// Stepwise homing process
CASE nTestStep OF
    0: // Await full power-up, start first stage home
        IF fbPower[4].PowerIsEnabled THEN
			 fbHome.Home(
					Position := fExpectedPosition,
					BufferMode := MC_BufferMode.MC_Aborting,
					HomeMode:=E_EpicsHomeCmd.HOME_VIA_HIGH
			);
            nTestStep := 1;
        END_IF
    1: // Simulate Forward Limit pulse (stage 1 complete)
        IF fbCamSwitchPulserSearch.Q THEN
            fbLimSwStatus[4].LimitForwardEnable := FALSE;
            fbCamSwitchPulserSearch.IN := FALSE;
            fbCamSwitchPulserSync.IN := TRUE;
            nTestStep := 2;
        END_IF
    2: // Release Forward Limit (simulate rising edge)
        IF fbCamSwitchPulserSync.Q THEN
            fbLimSwStatus[4].LimitForwardEnable := TRUE;
            nTestStep := 3;
        END_IF
    3: // When forward limit home is done, prepare for the home switch
        IF fbHome.LimHomeDone THEN
            fbCamSwitchPulserSearch.IN := TRUE;
            fbCamSwitchPulserSync.IN := FALSE;
            nTestStep := 4;
        END_IF
    4: // Simulate Home switch pulse
        IF fbCamSwitchPulserSearch.Q THEN
            fbLimSwStatus[4].LimitHome := TRUE;
            fbCamSwitchPulserSearch.IN := FALSE;
            fbCamSwitchPulserSync.IN := TRUE;
            nTestStep := 5;
        END_IF
    5: // Release Home switch
        IF fbCamSwitchPulserSync.Q THEN
            fbLimSwStatus[4].LimitHome := FALSE;
            nTestStep := 6;
        END_IF
    6: // Wait for homing full completion
        IF fbHome.Done THEN
            nTestStep := 7;
        END_IF
END_CASE

// Cyclic calls required for simulation and status updates
fbPower[4]();
fbHome();
fbCamSwitchPulserSearch();
fbCamSwitchPulserSync();
fbTestTimer();

// Finish test if homing is complete (step 7), or timeout
IF nTestStep = 7 THEN
    bCalibrated := fbHome.Done;
    AssertEquals_BOOL(
        Expected := TRUE,
        Actual := fbAxisRef[4].Status.Homed,
        Message := 'Axis not calibrated #1'
    );
    AssertEquals_LREAL(
        Delta := 0.001,
        Expected := fExpectedPosition,
        Actual := fbAxisRef[4].NcToPlc.ActPos,
        Message := 'Position is not the expected #2'
    );
    TEST_FINISHED();

ELSIF fbTestTimer.Q THEN
    AssertTrue(
        Condition := FALSE,
        Message := CONCAT('Timed out at step: ', TO_STRING(nTestStep))
    );
    TEST_FINISHED();
END_IF
END_METHOD

METHOD PRIVATE GivenHomeCmdHomeViaLowModeAndHomeSwPulseThenMoveToUserDefineOffset_Test5
VAR_INST
    fbHome : FB_HomeNC(
		AxisRef:=fbAxisRef[5],
		iLimSwStatus:=fbLimSwStatus[5],
		iMotionLogger:=fbMotionLogger[5]
	) := ( Mode := E_EpicsHomeCmd.HOME_VIA_LOW );
	
    fbTestTimer: TON := (IN:=TRUE, PT:=T#5S);
    fbCamSwitchPulserSearch: TON := (IN:=TRUE, PT:=T#500MS);
    fbCamSwitchPulserSync: TON := (PT:=T#1000MS);
    nTestStep : INT;
    fExpectedPosition : LREAL := 20.0;
    fActPosition : LREAL;
	bCalibrated: BOOL;
    // reset this when error or homeDone
    bHomingOverride : BOOL := TRUE;

END_VAR
TEST(__POUNAME());

// Cyclic status/logic blocks
fbLimSwStatus[5]();
fbMotionLogger[5]();

fbPower[5].Power(
    Enable := TRUE,
    Enable_Positive := bHomingOverride OR fbLimSwStatus[5].LimitForwardEnable,
    Enable_Negative := bHomingOverride OR fbLimSwStatus[5].LimitBackwardEnable,
    Override := 100.0
);

// State machine for homing by home switch
CASE nTestStep OF
    0: // Wait for power to enable before starting home sequence
        IF fbPower[5].PowerIsEnabled THEN
			 fbHome.Home(
					Position := fExpectedPosition,
					BufferMode := MC_BufferMode.MC_Aborting,
					HomeMode:=E_EpicsHomeCmd.HOME_VIA_LOW
			);
            nTestStep := 1;
        END_IF
    1: // Simulate cam switch pulse: set home limit
        IF fbCamSwitchPulserSearch.Q THEN
            fbLimSwStatus[5].LimitHome := TRUE;
            fbCamSwitchPulserSearch.IN := FALSE;
            fbCamSwitchPulserSync.IN := TRUE;
            nTestStep := 2;
        END_IF
    2: // Simulate sync pulse: clear home limit
        IF fbCamSwitchPulserSync.Q THEN
            fbLimSwStatus[5].LimitHome := FALSE;
            nTestStep := 3;
        END_IF
    3: // Wait for homing to complete
        IF fbHome.Done THEN
            nTestStep := 4;
        END_IF
    4:
        // No actions; test finishes in the assertion below
END_CASE

// Always cycle these for PLC logic to work
fbAxisRef[5].ReadStatus();
fbPower[5]();
fbHome();
fbCamSwitchPulserSearch();
fbCamSwitchPulserSync();
fbTestTimer();

// Assertions and test finish
IF nTestStep = 4 THEN
    bCalibrated := fbHome.Done;
    AssertEquals_BOOL(
        Expected := TRUE,
        Actual := fbAxisRef[5].Status.Homed,
        Message := 'Axis not calibrated #1'
    );
    AssertEquals_LREAL(
        Delta := 0.001,
        Expected := fExpectedPosition,
        Actual := fbAxisRef[5].NcToPlc.ActPos,
        Message := 'Position is not the expected #2'
    );
    TEST_FINISHED();

ELSIF fbTestTimer.Q THEN
    AssertTrue(
        Condition := FALSE,
        Message := CONCAT('Timed out at step: ', TO_STRING(nTestStep))
    );
    TEST_FINISHED();
END_IF
END_METHOD

METHOD PRIVATE GivenHomeCmdHomeViaLowModeBackwardSwPulseBeforeHomeSwPulseThenMoveToUserDefineOffset_Test6
VAR_INST
    fbHome : FB_HomeNC(
		AxisRef:=fbAxisRef[6],
		iLimSwStatus:=fbLimSwStatus[6],
		iMotionLogger:=fbMotionLogger[6]
	) := ( Mode:= E_EpicsHomeCmd.HOME_VIA_LOW );
	
    fbTestTimer: TON := (IN:=TRUE, PT:=T#5S);
    fbCamSwitchPulserSearch: TON := (IN:=TRUE, PT:=T#500MS);
    fbCamSwitchPulserSync: TON := (PT:=T#1000MS);
    nTestStep : INT;
    fExpectedPosition : LREAL := 20.0;
    fActPosition : LREAL;
	bCalibrated: BOOL;
    // reset this when error or homeDone
    bHomingOverride : BOOL := TRUE;

END_VAR
TEST(__POUNAME());

// Always call these each cycle for correct PLC scan semantics
fbAxisRef[6].ReadStatus();
fbLimSwStatus[6]();
fbMotionLogger[6]();

fbPower[6].Power(
    Enable := TRUE,
    Enable_Positive := bHomingOverride OR fbLimSwStatus[6].LimitForwardEnable,
    Enable_Negative := bHomingOverride OR fbLimSwStatus[6].LimitBackwardEnable,
    Override := 100.0
);

// State machine for negative (backward) limit then home
CASE nTestStep OF
    0: // Wait for power ready, then start home
        IF fbPower[6].PowerIsEnabled THEN
			 fbHome.Home(
					Position := fExpectedPosition,
					BufferMode := MC_BufferMode.MC_Aborting,
					HomeMode:=E_EpicsHomeCmd.HOME_VIA_LOW
			);
            nTestStep := 1;
        END_IF

    1: // Simulate cam pulse: deactivate backward limit
        IF fbCamSwitchPulserSearch.Q THEN
            fbLimSwStatus[6].LimitBackwardEnable := FALSE;
            fbCamSwitchPulserSearch.IN := FALSE;
            fbCamSwitchPulserSync.IN := TRUE;
            nTestStep := 2;
        END_IF

    2: // Reactivate backward limit on sync pulse
        IF fbCamSwitchPulserSync.Q THEN
            fbLimSwStatus[6].LimitBackwardEnable := TRUE;
            nTestStep := 3;
        END_IF

    3: // Wait for negative-limit home done, then prep second stage (home switch)
        IF fbHome.LimHomeDone THEN
            fbCamSwitchPulserSearch.IN := TRUE;
            fbCamSwitchPulserSync.IN := FALSE;
            nTestStep := 4;
        END_IF

    4: // Simulate home switch pulse
        IF fbCamSwitchPulserSearch.Q THEN
            fbLimSwStatus[6].LimitHome := TRUE;
            fbCamSwitchPulserSearch.IN := FALSE;
            fbCamSwitchPulserSync.IN := TRUE;
            nTestStep := 5;
        END_IF

    5: // Deactivate home switch after sync pulse
        IF fbCamSwitchPulserSync.Q THEN
            fbLimSwStatus[6].LimitHome := FALSE;
            nTestStep := 6;
        END_IF

    6: // Wait for full home sequence completion
        IF fbHome.Done THEN
            nTestStep := 7;
        END_IF

    7: // Test ends — handled below
END_CASE

// Cyclic calls
fbPower[6]();
fbHome();
fbCamSwitchPulserSearch();
fbCamSwitchPulserSync();
fbTestTimer();

// Assertion and finish logic
IF nTestStep = 7 THEN
    bCalibrated := fbHome.Done;

    AssertEquals_BOOL(
        Expected := TRUE,
        Actual := fbAxisRef[6].Status.Homed,
        Message := 'Axis not calibrated #1'
    );

    AssertEquals_LREAL(
        Delta := 0.001,
        Expected := fExpectedPosition,
        Actual := fbAxisRef[6].NcToPlc.ActPos,
        Message := 'Position is not the expected #2'
    );

    TEST_FINISHED();

ELSIF fbTestTimer.Q THEN
    AssertTrue(
        Condition := FALSE,
        Message := CONCAT('Timed out at step: ', TO_STRING(nTestStep))
    );
    TEST_FINISHED();
END_IF
END_METHOD

METHOD PRIVATE GivenHomeCmdLowLimitModeAndABackwardSwPulseThenHomeDoneAndPositionSetToUserDefineOffset_Test7
VAR_INST
    fbHome : FB_HomeNC(
		AxisRef:=fbAxisRef[7],
		iLimSwStatus:=fbLimSwStatus[7],
		iMotionLogger:=fbMotionLogger[7]
	) := ( Mode:= E_EpicsHomeCmd.LOW_LIMIT );
    fbTestTimer: TON := (IN:=TRUE, PT:=T#5S);
    fbCamSwitchPulserSearch: TON := (IN:=TRUE, PT:=T#500MS);
    fbCamSwitchPulserSync: TON := (PT:=T#1000MS);
    nTestStep : INT;
    fExpectedPosition : LREAL := 20.0;
    fActPosition : LREAL;
    bCalibrated: BOOL;
    // reset this when error or homeDone
    bHomingOverride : BOOL := TRUE;
END_VAR
TEST(__POUNAME());

// Cyclically called blocks
fbLimSwStatus[7]();
fbMotionLogger[7]();

fbPower[7].Power(
    Enable := TRUE,
    Enable_Positive := bHomingOverride OR fbLimSwStatus[7].LimitForwardEnable,
    Enable_Negative := bHomingOverride OR fbLimSwStatus[7].LimitBackwardEnable,
    Override := 100.0
);

// State machine for negative (backward) limit homing
CASE nTestStep OF
    0: // Wait for power enabled, then start homing
        IF fbPower[7].PowerIsEnabled THEN
			 fbHome.Home(
					Position := fExpectedPosition,
					BufferMode := MC_BufferMode.MC_Aborting,
					HomeMode:=E_EpicsHomeCmd.LOW_LIMIT
			);
            nTestStep := 1;
        END_IF

    1: // Simulate cam pulse to release backward limit
        IF fbCamSwitchPulserSearch.Q THEN
            fbLimSwStatus[7].LimitBackwardEnable := FALSE;
            fbCamSwitchPulserSearch.IN := FALSE;
            fbCamSwitchPulserSync.IN := TRUE;
            nTestStep := 2;
        END_IF

    2: // Simulate restoring backward limit
        IF fbCamSwitchPulserSync.Q THEN
            fbLimSwStatus[7].LimitBackwardEnable := TRUE;
            nTestStep := 3;
        END_IF

    3: // Wait for homing to complete
        IF fbHome.Done THEN
            nTestStep := 4;
        END_IF

    4: // Test ends; assertions below
END_CASE

// Always cycle axis status, home FB, cam pulsers, and timer
fbAxisRef[7].ReadStatus();
fbHome();
fbCamSwitchPulserSearch();
fbCamSwitchPulserSync();
fbTestTimer();

// Assertion and finish
IF nTestStep = 4 THEN
    bCalibrated := fbHome.Done;
    AssertEquals_BOOL(
        Expected := TRUE,
        Actual := fbAxisRef[7].Status.Homed,
        Message := 'Axis not calibrated #1'
    );
    AssertEquals_LREAL(
        Delta := 0.001,
        Expected := fExpectedPosition,
        Actual := fbAxisRef[7].NcToPlc.ActPos,
        Message := 'Position is not the expected #2'
    );
    TEST_FINISHED();

ELSIF fbTestTimer.Q THEN
    AssertTrue(
        Condition := FALSE,
        Message := CONCAT('Timed out at step: ', TO_STRING(nTestStep))
    );
    TEST_FINISHED();
END_IF
END_METHOD

METHOD PRIVATE GivenHomeCmdNoneModeThenSetHomeFlag_Test8
VAR_INST
    fbHome : FB_HomeNC(
		AxisRef:=fbAxisRef[8],
		iLimSwStatus:=fbLimSwStatus[8],
		iMotionLogger:=fbMotionLogger[8]
	):=(Mode:=E_EpicsHomeCmd.NONE);
    fbTestTimer: TON := (IN:=TRUE, PT:=T#5S);
    nTestStep : INT;
END_VAR
TEST(__POUNAME());

// Always call these each scan
fbLimSwStatus[8]();
fbMotionLogger[8]();

// State machine for basic home sequence
CASE nTestStep OF
    0: // Enable axis power
        fbPower[8].Power(
            Enable := TRUE,
            Enable_Positive := fbLimSwStatus[8].LimitForwardEnable,
            Enable_Negative := fbLimSwStatus[8].LimitBackwardEnable,
            Override := 100.0
        );
        nTestStep := 1;

    1: // Wait for power to come up, then issue Home command
        IF fbPower[8].PowerIsEnabled THEN
			 fbHome.Home(
					Position := 0.0,
					BufferMode := MC_BufferMode.MC_Aborting,
					HomeMode:=E_EpicsHomeCmd.NONE
			);
            nTestStep := 2;
        END_IF

    2: // Wait for homing to finish
        IF fbHome.Done THEN
            nTestStep := 3;
        END_IF

    3: // Test ends; assertion and finish below
END_CASE

// Required cyclic calls
fbPower[8]();
fbHome();
fbTestTimer(IN := TRUE);

// Assertion & finish logic
IF nTestStep = 3 THEN
    // You may add validation here (homed position, calibrated flag, etc.) if required
    TEST_FINISHED();
ELSIF fbTestTimer.Q THEN
    AssertTrue(
        Condition := FALSE,
        Message := CONCAT('Timed out at step: ', TO_STRING(nTestStep))
    );
    TEST_FINISHED();
END_IF
END_METHOD

METHOD PRIVATE GivenHomeCmdSetToHighLimitAndHighLimitPulseThenSetHomeDoneAndPositionToUserDefineOffset_Test9
VAR_INST
    fbHome : FB_HomeNC(
		AxisRef:=fbAxisRef[9],
		iLimSwStatus:=fbLimSwStatus[9],
		iMotionLogger:=fbMotionLogger[9]
	):=(Mode:=E_EpicsHomeCmd.HIGH_LIMIT);
	
    fbTestTimer: TON := (IN:=TRUE, PT:=T#5S);
    fbCamSwitchPulserSearch: TON := (IN:=TRUE, PT:=T#500MS);
    fbCamSwitchPulserSync: TON := (PT:=T#1000MS);
    nTestStep : INT;
    fExpectedPosition : LREAL := 20.0;
    fActPosition : LREAL;
    bCalibrated: BOOL;
    // reset this when error or homeDone
    bHomingOverride : BOOL := TRUE;
END_VAR
TEST(__POUNAME());

// Cyclic calls: always invoked every scan
fbLimSwStatus[9]();
fbMotionLogger[9]();
fbPower[9].Power(
    Enable := TRUE,
    Enable_Positive := bHomingOverride OR fbLimSwStatus[9].LimitForwardEnable,
    Enable_Negative := bHomingOverride OR fbLimSwStatus[9].LimitBackwardEnable,
    Override := 100.0
);

// Homing state machine
CASE nTestStep OF
    0: // Wait for power enabled, then start homing command
        IF fbPower[9].PowerIsEnabled THEN
			 fbHome.Home(
					Position := fExpectedPosition,
					BufferMode := MC_BufferMode.MC_Aborting,
					HomeMode:=E_EpicsHomeCmd.HIGH_LIMIT
			);
            nTestStep := 1;
        END_IF

    1: // Simulate cam pulse to clear forward limit
        IF fbCamSwitchPulserSearch.Q THEN
            fbLimSwStatus[9].LimitForwardEnable := FALSE;
            fbCamSwitchPulserSearch.IN := FALSE;
            fbCamSwitchPulserSync.IN := TRUE;
            nTestStep := 2;
        END_IF

    2: // Simulate restoring forward limit
        IF fbCamSwitchPulserSync.Q THEN
            fbLimSwStatus[9].LimitForwardEnable := TRUE;
            nTestStep := 3;
        END_IF

    3: // Wait for homing to complete
        IF fbHome.Done THEN
            nTestStep := 4;
        END_IF

    4: // Test ends, assertions handled below
END_CASE

// Always called each scan
fbAxisRef[9].ReadStatus();
fbHome();
fbCamSwitchPulserSearch();
fbCamSwitchPulserSync();
fbTestTimer();

// Assertion and finish
IF nTestStep = 4 THEN
    bCalibrated := fbHome.Done;
    AssertEquals_BOOL(
        Expected := TRUE,
        Actual := fbAxisRef[9].Status.Homed,
        Message := 'Axis not calibrated #1'
    );
    AssertEquals_LREAL(
        Delta := 0.001,
        Expected := fExpectedPosition,
        Actual := fbAxisRef[9].NcToPlc.ActPos,
        Message := 'Position is not the expected #2'
    );
    TEST_FINISHED();

ELSIF fbTestTimer.Q THEN
    AssertTrue(
        Condition := FALSE,
        Message := CONCAT('Timed out at step: ', TO_STRING(nTestStep))
    );
    TEST_FINISHED();
END_IF
END_METHOD

METHOD PRIVATE GivenMoveCmdNegativeBacklashCompensationActiveThenReverseMoveIsCompensated_Test10
VAR_INST
    // Subjects under tests
    fbBacklashCompensation : FB_BacklashCompensationNC(AxisRef := fbAxisRef[10],  iMotionLogger:= fbMotionLogger[10]);
    fbMoveAbsolute : FB_MoveAbsoluteNC(AxisRef := fbAxisRef[10],  iMotionLogger:= fbMotionLogger[10]);
    // Backalsh is testing on simulated NC axis in Homing and PTP
    fbTestTimer : TON := (PT := T#5S, IN := TRUE);
    nTestStep : INT;;

END_VAR
TEST(__POUNAME());

// Must be called cyclically
fbPower[10].Power(
    Enable := TRUE,
    Enable_Positive := fbLimSwStatus[10].LimitForwardEnable,
    Enable_Negative := fbLimSwStatus[10].LimitBackwardEnable,
    Override := 100
);

CASE nTestStep OF
    // Enable compensation, but status should still be OFF initially
    0:
        fbBacklashCompensation.EnableBacklashCompensation(UserEnable := TRUE, Compensation := -4.0);
        nTestStep := 1;
	1:
		fbBacklashCompensation.BacklashCompensation(Enable := TRUE, RampVelo := 10.0);
		nTestStep := 2;
    2:
        AssertTrue(
            Condition := fbBacklashCompensation.Status,
            Message := 'Backlash compensation must be enabled #2'
        );
        nTestStep := 3;

    // Start negative move (direction should not apply backlash compensation here)
    3:
        IF fbPower[10].PowerIsEnabled THEN
            fbMoveAbsolute.MoveAbsolute(
                Position := -10.0,
                Velocity := 100,
                Acceleration := 200,
                Deceleration := 200
            );
            nTestStep := 4;
        END_IF

    // Assert compensation does not apply after negative move
   4:
        IF fbMoveAbsolute.Done THEN
            AssertTrue(
                Condition := (fbAxisRef[10].NcToPlc.ActPos - fbAxisRef[10].NcToPlc.ActPosWithoutPosCorrection) = 0,
                Message := 'No Backlash compensation in this direction #3'
            );
            nTestStep := 5;
        END_IF

    // Start reverse move (should apply backlash compensation)
   5:
        fbMoveAbsolute.MoveAbsolute(
            Position := 20.0,
            Velocity := 100,
            Acceleration := 200,
            Deceleration := 200
        );
        nTestStep := 6;

    // Assert compensation is applied after reverse move
   6:
        IF fbMoveAbsolute.Done THEN
            AssertTrue(
                Condition := (fbAxisRef[10].NcToPlc.ActPos - fbAxisRef[10].NcToPlc.ActPosWithoutPosCorrection) = 4,
                Message := 'Current backlash must be 4 #4'
            );
            nTestStep := 7;
        END_IF

END_CASE

// Required cyclic calls
fbBacklashCompensation();
fbMoveAbsolute();
fbTestTimer();

// Final assertion and finish
IF nTestStep = 7 THEN
    AssertTrue(
        Condition := fbBacklashCompensation.Status,
        Message := 'Backlash compensation must stay enabled after absolute move #5'
    );
    TEST_FINISHED();

ELSIF fbTestTimer.Q THEN
    AssertTrue(
        Condition := FALSE,
        Message := CONCAT('Timed out at step: ', TO_STRING(nTestStep))
    );
    TEST_FINISHED();
END_IF
END_METHOD

METHOD PRIVATE GivenMoveCmdPositiveBacklashCompensationActiveThenReverseMoveIsCompensated_Test11
VAR_INST
    // Subjects under test
    fbBacklashCompensation : FB_BacklashCompensationNC(AxisRef := fbAxisRef[11],  iMotionLogger:= fbMotionLogger[11]);
	fbMoveAbsolute : FB_MoveAbsoluteNC(AxisRef := fbAxisRef[11],  iMotionLogger:= fbMotionLogger[11]);
    // Backalsh is testing on simulated NC axis in Homing and PTP
    fbTestTimer : TON := (PT := T#5S, IN := TRUE);
    nTestStep : INT;

    


END_VAR
TEST(__POUNAME());

// Must be called cyclically
fbPower[11].Power(
    Enable := TRUE,
    Enable_Positive := fbLimSwStatus[11].LimitForwardEnable,
    Enable_Negative := fbLimSwStatus[11].LimitBackwardEnable,
    Override := 100
);

CASE nTestStep OF
    // Enable compensation, but status should still be OFF initially
    0:
        fbBacklashCompensation.EnableBacklashCompensation(UserEnable := TRUE, Compensation := 4.0);
        nTestStep := 1;
	1:
		fbBacklashCompensation.BacklashCompensation(Enable := TRUE, RampVelo := 10.0);
		nTestStep := 2;
    2:
        AssertTrue(
            Condition := fbBacklashCompensation.Status,
            Message := 'Backlash compensation must be enabled #2'
        );
        nTestStep := 3;

    // Start negative move (direction should not apply backlash compensation here)
    3:
        IF fbPower[11].PowerIsEnabled THEN
            fbMoveAbsolute.MoveAbsolute(
                Position :=50.0,
                Velocity := 100,
                Acceleration := 200,
                Deceleration := 200
            );
            nTestStep := 4;
        END_IF

    // Assert compensation does not apply after negative move
   4:
        IF fbMoveAbsolute.Done THEN
            AssertTrue(
                Condition := (fbAxisRef[11].NcToPlc.ActPos - fbAxisRef[11].NcToPlc.ActPosWithoutPosCorrection) = 0,
                Message := 'No Backlash compensation in this direction #3'
            );
            nTestStep := 5;
        END_IF

    // Start reverse move (should apply backlash compensation)
   5:
        fbMoveAbsolute.MoveAbsolute(
            Position := 25.0,
            Velocity := 100,
            Acceleration := 200,
            Deceleration := 200
        );
        nTestStep := 6;

    // Assert compensation is applied after reverse move
   6:
        IF fbMoveAbsolute.Done THEN
            AssertTrue(
                Condition := (fbAxisRef[11].NcToPlc.ActPos - fbAxisRef[11].NcToPlc.ActPosWithoutPosCorrection) = 4,
                Message := 'Current backlash must be 4 #4'
            );
            nTestStep := 7;
        END_IF

END_CASE

// Required cyclic calls
fbBacklashCompensation();
fbMoveAbsolute();
fbTestTimer();

// Final assertion and finish
IF nTestStep = 7 THEN
    AssertTrue(
        Condition := fbBacklashCompensation.Status,
        Message := 'Backlash compensation must stay enabled after absolute move #5'
    );
    TEST_FINISHED();

ELSIF fbTestTimer.Q THEN
    AssertTrue(
        Condition := FALSE,
        Message := CONCAT('Timed out at step: ', TO_STRING(nTestStep))
    );
    TEST_FINISHED();
END_IF
END_METHOD

METHOD PRIVATE GivenPowerIsEnabledAbsoluteMoveIfResetThenMoveIsAbortedAndResetDoneIsRetained_Test16
VAR_INST
    // Subjects under test
    fbMoveAbsolute : FB_MoveAbsoluteNC(AxisRef := fbAxisRef[16], iMotionLogger:= fbMotionLogger[16]);
    fbReset : FB_ResetNC(AxisRef := fbAxisRef[16], iMotionLogger:= fbMotionLogger[16]);
    fbTestTimer : TON := (PT := T#3S, IN := TRUE);
    fbInMotionTimer : TON := (PT := T#1S, IN := FALSE);
    nTestStateStep : INT;
END_VAR
TEST(__POUNAME());

// Cyclic power logic
fbPower[16].Power(
    Enable := TRUE,
    Enable_Positive := fbLimSwStatus[16].LimitForwardEnable,
    Enable_Negative := fbLimSwStatus[16].LimitBackwardEnable,
    Override := 100
);

// State machine for move + reset abort
CASE nTestStateStep OF
    0: // Wait for axis power before starting move
        IF fbPower[16].PowerIsEnabled THEN
            nTestStateStep := 1;
        END_IF

    1: // Issue move absolute
        fbMoveAbsolute.MoveAbsolute(
            Position := 100,
            Velocity := 100,
            Acceleration := 50,
            Deceleration := 50
        );
        nTestStateStep := 2;

    2: // Wait for axis to become busy; start timer
        IF fbMoveAbsolute.Busy THEN
            fbInMotionTimer.IN := TRUE;
            nTestStateStep := 3;
        END_IF

    3: // When timer elapses, send Reset to abort move
        IF fbInMotionTimer.Q THEN
            fbReset.Reset();
            fbInMotionTimer.IN := FALSE;
            nTestStateStep := 4;
        END_IF

    4: // Wait for reset to be done (move abort completion)
        IF fbReset.Done THEN
            nTestStateStep := 5;
        END_IF
END_CASE

// Cyclic calls for status and timers
fbInMotionTimer();
fbAxisRef[16].ReadStatus();
fbMoveAbsolute();
fbReset();
fbTestTimer();

// Assertion and finish logic
IF nTestStateStep = 5 THEN
    AssertTrue(
        Condition := fbMoveAbsolute.Aborted,
        Message := 'Expected CommandAborted'
    );
    AssertTrue(
        Condition := fbReset.Done,
        Message := 'Expected Reset.Done'
    );
    AssertFalse(
        Condition := fbReset.Busy,
        Message := 'Expected Reset not busy'
    );
    TEST_FINISHED();

ELSIF fbTestTimer.Q THEN
    AssertTrue(
        Condition := FALSE,
        Message := CONCAT('Timed out at step: ', TO_STRING(nTestStateStep))
    );
    TEST_FINISHED();
END_IF
END_METHOD

METHOD PRIVATE GivenPowerIsEnabledAndAbsoluteMoveStartedIfHaltSignalThenMoveIsAbortedAndHaltDoneIsRetained_Test15
VAR_INST
    // Subjects under test
    fbMoveAbsolute : FB_MoveAbsoluteNC(AxisRef := fbAxisRef[15], iMotionLogger:= fbMotionLogger[15]);
    fbHalt : FB_HaltNC(AxisRef := fbAxisRef[15], iMotionLogger:= fbMotionLogger[15]);
    fbTestTimer : TON := (PT := T#3S, IN := TRUE);
    fbInMotionTimer : TON := (PT := T#1S, IN := FALSE);
    nTestStateStep : INT;;
END_VAR
TEST(__POUNAME());

// Always called per scan
fbPower[15].Power(
    Enable := TRUE,
    Enable_Positive := fbLimSwStatus[15].LimitForwardEnable,
    Enable_Negative := fbLimSwStatus[15].LimitBackwardEnable,
    Override := 100
);

// State machine for move + halt
CASE nTestStateStep OF
    0 : // Wait for power-up before starting move
        IF fbPower[15].PowerIsEnabled THEN
            nTestStateStep := 1;
        END_IF

    1 : // Start move
        fbMoveAbsolute.MoveAbsolute(
            Position := 100,
            Velocity := 100,
            Acceleration := 50,
            Deceleration := 50
        );
        nTestStateStep := 2;

    2 : // Wait until move system is busy, then start in-motion timer
        IF fbMoveAbsolute.Busy THEN
            fbInMotionTimer.IN := TRUE;
            nTestStateStep := 3;
        END_IF

    3 : // When timer triggers, send Halt
        IF fbInMotionTimer.Q THEN
            fbHalt.Halt(
                Deceleration := 100,
                Jerk := 0
            );
            fbInMotionTimer.IN := FALSE;
            nTestStateStep := 4;
        END_IF

    4 : // Wait for halt done (move abort confirmation)
        IF fbHalt.Done THEN
            nTestStateStep := 5;
        END_IF

    5 : // Test ends; assertions below
        // (do nothing)
END_CASE

// Cyclic calls
fbTestTimer();
fbInMotionTimer();
fbAxisRef[15].ReadStatus();
fbMoveAbsolute();
fbHalt();

// Test result and finish logic
IF nTestStateStep = 5 THEN
    AssertTrue(
        Condition := fbMoveAbsolute.Aborted,
        Message := 'Expected CommandAborted'
    );
    AssertTrue(
        Condition := fbHalt.Done,
        Message := 'Expected Done'
    );
    AssertFalse(
        Condition := fbHalt.Busy,
        Message := 'Expected not busy'
    );
    TEST_FINISHED();

ELSIF fbTestTimer.Q THEN
    AssertTrue(
        Condition := FALSE,
        Message := CONCAT('Timed out at step: ', TO_STRING(nTestStateStep))
    );
    TEST_FINISHED();
END_IF
END_METHOD

METHOD PRIVATE GivenPowerIsEnabledAndCompletedAbsoluteMoveThenMoveAbsoluteDoneStatusRetained_Test14
VAR_INST
    fbMoveAbsolute : FB_MoveAbsoluteNC(AxisRef := fbAxisRef[14], iMotionLogger:= fbMotionLogger[14]);
    nTestStateStep : INT;
    fbTestTimer : TON := (PT := T#3S, IN := TRUE);
    fExpectedPosition: LREAL := 50.0;
END_VAR
TEST(__POUNAME());

// Always call required power block
fbPower[14].Power(
    Enable := TRUE,
    Enable_Positive := fbLimSwStatus[14].LimitForwardEnable,
    Enable_Negative := fbLimSwStatus[14].LimitBackwardEnable,
    Override := 100
);

// Stepwise state machine for the move
CASE nTestStateStep OF
    0 : // Wait for power-on before starting move
        IF fbPower[14].PowerIsEnabled THEN
            nTestStateStep := 1;
        END_IF

    1 : // Issue Move Absolute command
        fbMoveAbsolute.MoveAbsolute(
            Position := fExpectedPosition,   // Substituted value for clarity
            Velocity := 500,
            Acceleration := 1000,
            Deceleration := 1000
        );
        nTestStateStep := 2;

    2 : // Wait until move finishes
        IF fbMoveAbsolute.Done THEN
            nTestStateStep := 3;
        END_IF
END_CASE

// Cyclically called per scan
fbTestTimer();
fbAxisRef[14].ReadStatus();
fbMoveAbsolute();

// Final assertion and test finish
IF nTestStateStep = 3 THEN
    AssertEquals_LREAL(
        Delta := 0.001,
        Expected := fExpectedPosition,
        Actual := fbAxisRef[14].NcToPlc.ActPos,
        Message := 'Position is not the expected #1'
    );
    TEST_FINISHED();

ELSIF fbTestTimer.Q THEN
    AssertTrue(
        Condition := FALSE,
        Message := CONCAT('Timed out at step: ', TO_STRING(nTestStateStep))
    );
    TEST_FINISHED();
END_IF
END_METHOD

END_FUNCTION_BLOCK

// ---- Test/NC/FB_MotionAxisNC_Test.TcPOU
FUNCTION_BLOCK FB_MotionAxisNC_Test EXTENDS FB_TestSuite
VAR
	fbAxisRef : AXIS_REF;
	fbMotionLogger : FB_MotionLogger_TestDouble;
    fbHome : FB_HomeNC_TestDouble;
    fbHalt : FB_HaltNC_TestDouble;
    fbPower : FB_PowerNC_TestDouble;
    fbReset : FB_ResetNC_TestDouble;
    fbMoveAbsolute : FB_MoveAbsoluteNC_TestDouble;
    fbReadParameter : FB_ReadParameterNC_TestDouble;
    fbWriteParameter  : FB_WriteParameterNC_TestDouble;
    fbParamSaveRestore: FB_ParamSaveRestoreNC_TestDouble;
    fbEncoderScaling : FB_EncoderScalingNC_TestDouble;
    fbAxisStatus : FB_AxisStatusNC_TestDouble;
    fbBacklashCompensation : FB_BacklashCompensationNC_TestDouble;
END_VAR

GivenAllMCBlockErrorConditionThenPowerErrorHasHigherPriority();

METHOD PRIVATE GivenAllMCBlockErrorConditionThenPowerErrorHasHigherPriority
VAR_INST
    // subject under test
    // subject under test
    fbMotionAxis : FB_MotionAxisNC(  	
		AxisRef :=fbAxisRef,
		iMotionLogger := fbMotionLogger,
		iHome := fbHome,
        iHalt := fbHalt,
        iPower := fbPower,
        iReset := fbReset,
        iMoveAbsolute := fbMoveAbsolute,
        iReadParameter := fbReadParameter,
        iWriteParameter  := fbWriteParameter,
        iParamsSaveRestore:= fbParamSaveRestore,
        iEncoderScaling := fbEncoderScaling,
        iBacklashCompensation := fbBacklashCompensation
	);
bExpectedAxisError :BOOL := TRUE;
nExpectedErrorId: UDINT;
END_VAR
TEST(__POUNAME());
// ----- Power: Highest priority -----
fbHome.Error := TRUE;
fbHalt.Error := TRUE;
fbPower.Error := TRUE;
fbReset.Error := TRUE;
fbMoveAbsolute.Error := TRUE;
fbReadParameter.Error := TRUE;
fbWriteParameter.Error := TRUE;
fbParamSaveRestore.Error := TRUE;
fbBacklashCompensation.Error := TRUE;

fbMotionAxis();

AssertTrue(
    Condition := fbMotionAxis.Status.bError,
    Message   := 'Prioritized and generalized Error must be set #1'
);
AssertEquals_UDINT(
    Expected := 18000,
    Actual   := fbMotionAxis.Status.nErrorID,
    Message  := 'Prioritized error Id must be 18000 #2'
);

// ----- Halt: Second -----
fbPower.Error := FALSE;
fbHalt.Error := TRUE;
fbHome.Error := TRUE;
fbReset.Error := TRUE;
fbMoveAbsolute.Error := TRUE;
fbReadParameter.Error := TRUE;
fbWriteParameter.Error := TRUE;
fbParamSaveRestore.Error := TRUE;
fbBacklashCompensation.Error := TRUE;

fbMotionAxis();

AssertTrue(
    Condition := fbMotionAxis.Status.bError,
    Message   := 'Prioritized and generalized Error must be set #3'
);
AssertEquals_UDINT(
    Expected := 19000,
    Actual   := fbMotionAxis.Status.nErrorID,
    Message  := 'Prioritized error Id must be 19000 #4'
);

// ----- Reset: Third -----
fbPower.Error := FALSE;
fbHalt.Error := FALSE;
fbReset.Error := TRUE;
fbHome.Error := TRUE;
fbMoveAbsolute.Error := TRUE;
fbReadParameter.Error := TRUE;
fbWriteParameter.Error := TRUE;
fbParamSaveRestore.Error := TRUE;
fbBacklashCompensation.Error := TRUE;

fbMotionAxis();

AssertTrue(
    Condition := fbMotionAxis.Status.bError,
    Message   := 'Prioritized and generalized Error must be set #5'
);
AssertEquals_UDINT(
    Expected := 20000,
    Actual   := fbMotionAxis.Status.nErrorID,
    Message  := 'Prioritized error Id must be 20000 #6'
);

// ----- BacklashCompensation: Fourth -----
fbPower.Error := FALSE;
fbHalt.Error := FALSE;
fbReset.Error := FALSE;
fbBacklashCompensation.Error := TRUE;
fbHome.Error := TRUE;
fbMoveAbsolute.Error := TRUE;
fbReadParameter.Error := TRUE;
fbWriteParameter.Error := TRUE;
fbParamSaveRestore.Error := TRUE;

fbMotionAxis();

AssertTrue(
    Condition := fbMotionAxis.Status.bError,
    Message   := 'Prioritized and generalized Error must be set #7'
);
AssertEquals_UDINT(
    Expected := 21000,
    Actual   := fbMotionAxis.Status.nErrorID,
    Message  := 'Prioritized error Id must be 21000 #8'
);

// ----- MoveAbsolute: Fifth -----
fbBacklashCompensation.Error := FALSE;
fbMoveAbsolute.Error := TRUE;
fbPower.Error := FALSE;
fbHalt.Error := FALSE;
fbReset.Error := FALSE;
fbHome.Error := TRUE;
fbReadParameter.Error := TRUE;
fbWriteParameter.Error := TRUE;
fbParamSaveRestore.Error := TRUE;

fbMotionAxis();

AssertTrue(
    Condition := fbMotionAxis.Status.bError,
    Message   := 'Prioritized and generalized Error must be set #9'
);
AssertEquals_UDINT(
    Expected := 22000,
    Actual   := fbMotionAxis.Status.nErrorID,
    Message  := 'Prioritized error Id must be 22000 #10'
);

// ----- Home: Sixth -----
fbMoveAbsolute.Error := FALSE;
fbHome.Error := TRUE;
fbPower.Error := FALSE;
fbHalt.Error := FALSE;
fbReset.Error := FALSE;
fbBacklashCompensation.Error := FALSE;
fbReadParameter.Error := TRUE;
fbWriteParameter.Error := TRUE;
fbParamSaveRestore.Error := TRUE;

fbMotionAxis();

AssertTrue(
    Condition := fbMotionAxis.Status.bError,
    Message   := 'Prioritized and generalized Error must be set #11'
);
AssertEquals_UDINT(
    Expected := 23000,
    Actual   := fbMotionAxis.Status.nErrorID,
    Message  := 'Prioritized error Id must be 23000 #12'
);

// ----- ReadParameter: Eighth -----
fbHome.Error := FALSE;
fbReadParameter.Error := TRUE;
fbWriteParameter.Error := TRUE;
fbPower.Error := FALSE;
fbHalt.Error := FALSE;
fbReset.Error := FALSE;
fbBacklashCompensation.Error := FALSE;
fbMoveAbsolute.Error := FALSE;
fbParamSaveRestore.Error := TRUE;

fbMotionAxis();

AssertTrue(
    Condition := fbMotionAxis.Status.bError,
    Message   := 'Prioritized and generalized Error must be set #13'
);
AssertEquals_UDINT(
    Expected := 25000,
    Actual   := fbMotionAxis.Status.nErrorID,
    Message  := 'Prioritized error Id must be 25000 #14'
);

// ----- WriteParameter: Ninth -----
fbReadParameter.Error := FALSE;
fbWriteParameter.Error := TRUE;
fbPower.Error := FALSE;
fbHalt.Error := FALSE;
fbReset.Error := FALSE;
fbBacklashCompensation.Error := FALSE;
fbMoveAbsolute.Error := FALSE;
fbHome.Error := FALSE;
fbParamSaveRestore.Error := TRUE;

fbMotionAxis();

AssertTrue(
    Condition := fbMotionAxis.Status.bError,
    Message   := 'Prioritized and generalized Error must be set #15'
);
AssertEquals_UDINT(
    Expected := 26000,
    Actual   := fbMotionAxis.Status.nErrorID,
    Message  := 'Prioritized error Id must be 26000 #16'
);

// ----- ParamSaveRestore: Tenth -----
fbWriteParameter.Error := FALSE;
fbParamSaveRestore.Error := TRUE;
fbPower.Error := FALSE;
fbHalt.Error := FALSE;
fbReset.Error := FALSE;
fbBacklashCompensation.Error := FALSE;
fbMoveAbsolute.Error := FALSE;
fbHome.Error := FALSE;
fbReadParameter.Error := FALSE;

fbMotionAxis();

AssertTrue(
    Condition := fbMotionAxis.Status.bError,
    Message   := 'Prioritized and generalized Error must be set #17'
);
AssertEquals_UDINT(
    Expected := 27000,
    Actual   := fbMotionAxis.Status.nErrorID,
    Message  := 'Prioritized error Id must be 27000 #18'
);

TEST_FINISHED();
END_METHOD

END_FUNCTION_BLOCK

// ---- Test/TestDouble/FB_HaltNC_TestDouble.TcPOU
FUNCTION_BLOCK FB_HaltNC_TestDouble IMPLEMENTS  I_Halt
VAR
    bError : BOOL;
    nErrorID : UDINT := 19000;
END_VAR

PROPERTY Aborted : BOOL
GET
END_GET
END_PROPERTY

PROPERTY Active : BOOL
GET
Active := TRUE;
END_GET
END_PROPERTY

PROPERTY Busy : BOOL
GET
END_GET
END_PROPERTY

METHOD ClearStatus
END_METHOD

PROPERTY CommandHalt : BOOL
SET
END_SET
END_PROPERTY

PROPERTY Done : BOOL
GET
END_GET
END_PROPERTY

PROPERTY Error : BOOL
GET
Error := bError;
END_GET
SET
bError := Error;
END_SET
END_PROPERTY

PROPERTY ErrorID : UDINT
GET
ErrorId := nErrorID;
END_GET
SET
nErrorId := ErrorID;
END_SET
END_PROPERTY

METHOD Halt
VAR_INPUT
    Deceleration	: LREAL := 0;
    Jerk	: LREAL := 0;
    BufferMode	: MC_BufferMode := MC_BufferMode.MC_Aborting;
END_VAR
END_METHOD

PROPERTY Message : T_MAXSTRING
GET
END_GET
END_PROPERTY

END_FUNCTION_BLOCK

// ---- Test/TestDouble/FB_ResetNC_TestDouble.TcPOU
FUNCTION_BLOCK FB_ResetNC_TestDouble IMPLEMENTS  I_Reset
VAR
    bError : BOOL;
    nErrorID : UDINT := 20000;
END_VAR

PROPERTY Aborted : BOOL
GET
END_GET
END_PROPERTY

PROPERTY Active : BOOL
GET
Active := TRUE;
END_GET
END_PROPERTY

PROPERTY Busy : BOOL
GET
END_GET
END_PROPERTY

METHOD ClearStatus
END_METHOD

PROPERTY Done : BOOL
GET
END_GET
END_PROPERTY

PROPERTY Error : BOOL
GET
Error := bError;
END_GET
SET
bError := Error;
END_SET
END_PROPERTY

PROPERTY ErrorID : UDINT
GET
ErrorId := nErrorID;
END_GET
SET
nErrorId := ErrorID;
END_SET
END_PROPERTY

PROPERTY Message : T_MAXSTRING
GET
END_GET
END_PROPERTY

METHOD Reset
END_METHOD

END_FUNCTION_BLOCK

// ---- Test/TestDouble/FB_MoveAbsoluteNC_TestDouble.TcPOU
FUNCTION_BLOCK FB_MoveAbsoluteNC_TestDouble IMPLEMENTS I_MoveABsolute
VAR
    bError : BOOL;
    nErrorID : UDINT := 22000;
END_VAR

PROPERTY Aborted : BOOL
GET
END_GET
END_PROPERTY

PROPERTY Active : BOOL
GET
END_GET
END_PROPERTY

PROPERTY Busy : BOOL
GET
END_GET
END_PROPERTY

{warning 'Add method implementation '}
METHOD CLearStatus
END_METHOD

PROPERTY CommandMoveAbsolute : BOOL
SET
END_SET
END_PROPERTY

PROPERTY Done : BOOL
GET
END_GET
END_PROPERTY

PROPERTY Error : BOOL
GET
Error := bError;
END_GET
SET
bError := Error;
END_SET
END_PROPERTY

PROPERTY ErrorID : UDINT
GET
ErrorId := nErrorID;
END_GET
SET
nErrorId := ErrorID;
END_SET
END_PROPERTY

PROPERTY Message : T_MAXSTRING
GET
END_GET
END_PROPERTY

METHOD MoveAbsolute
VAR_INPUT
    Position	: LREAL;
    Velocity	: LREAL;
    Acceleration	: LREAL := 0;
    Deceleration	: LREAL := 0;
    Jerk	: LREAL := 0;
    BufferMode	: MC_BufferMode := MC_BufferMode.MC_Aborting;
END_VAR
END_METHOD

END_FUNCTION_BLOCK

// ---- Test/TestDouble/FB_ParamSaveRestoreNC_TestDouble.TcPOU
FUNCTION_BLOCK FB_ParamSaveRestoreNC_TestDouble IMPLEMENTS I_ParamsSaveRestore
VAR
    bError : BOOL;
    nErrorID : UDINT := 27000;
END_VAR

PROPERTY Aborted : BOOL
GET
END_GET
END_PROPERTY

PROPERTY Active : BOOL
GET
END_GET
END_PROPERTY

PROPERTY Busy : BOOL
GET
END_GET
END_PROPERTY

PROPERTY Done : BOOL
GET
END_GET
END_PROPERTY

PROPERTY Error : BOOL
GET
Error := bError;
END_GET
SET
bError := Error;
END_SET
END_PROPERTY

PROPERTY ErrorID : UDINT
GET
ErrorId := nErrorID;
END_GET
SET
nErrorId := ErrorID;
END_SET
END_PROPERTY

PROPERTY Message : T_MAXSTRING
GET
END_GET
END_PROPERTY

METHOD RestoreAxisParams
END_METHOD

METHOD SaveAxisParams
VAR_INPUT
    Enable	: BOOL;
END_VAR
END_METHOD

PROPERTY SavedPosition : LREAL
GET
END_GET
END_PROPERTY

END_FUNCTION_BLOCK

// ---- Test/TestDouble/FB_MotionInterlocksLimSw_TestDouble.TcPOU
FUNCTION_BLOCK FB_MotionInterlocksLimSw_TestDouble IMPLEMENTS I_MotionInterlocks
VAR
END_VAR

METHOD AxisStatus
VAR_INPUT
    HomeBusy	: BOOL;
    PositiveDirection	: BOOL;
    NegativeDirection	: BOOL;
END_VAR
END_METHOD

METHOD DriveCommands
VAR_INPUT
    MoveEnable: BOOL;
    NewMoveReq : BOOL;
END_VAR
END_METHOD

PROPERTY Error : BOOL
GET
END_GET
END_PROPERTY

PROPERTY ErrorID : UDINT
GET
END_GET
END_PROPERTY

{warning 'Add property implementation'}
PROPERTY HomeSensor : BOOL
GET
END_GET
END_PROPERTY

PROPERTY InterlockEvent : BOOL
GET
END_GET
END_PROPERTY

PROPERTY LimHome : BOOL
GET
END_GET
END_PROPERTY

PROPERTY Message : T_MAXSTRING
GET
END_GET
END_PROPERTY

PROPERTY MoveBackwardEnabled : BOOL
GET
END_GET
END_PROPERTY

PROPERTY MoveForwardEnabled : BOOL
GET
END_GET
END_PROPERTY

PROPERTY MoveOk : BOOL
GET
END_GET
END_PROPERTY

PROPERTY PowerEnabled : BOOL
GET
END_GET
END_PROPERTY

METHOD Reset
END_METHOD

PROPERTY Warning : BOOL
GET
END_GET
END_PROPERTY

END_FUNCTION_BLOCK

// ---- Test/TestDouble/FB_PersistentDataStorage_TestDouble.TcPOU
FUNCTION_BLOCK FB_PersistentDataStorage_TestDouble IMPLEMENTS I_PersistentDataStorage
VAR
END_VAR

{warning 'Add property implementation'}
PROPERTY TriggerWriteOfPersistentData : BOOL
GET
END_GET
SET
END_SET
END_PROPERTY

END_FUNCTION_BLOCK
